FUNCTION IsValidMetadatum : BOOL
VAR_INPUT
	Metadatum : I_Metadatum;
END_VAR

IsValidMetadatum := Metadatum <> 0;

END_FUNCTION

(* stored: Version 1.1.0.1, ProductVersion 3.1.4024.12
   POU IsValidMetadatum: Id {5d7b0806-07d4-0466-38a3-7d4f521ef374}, SpecialFunc None *)
